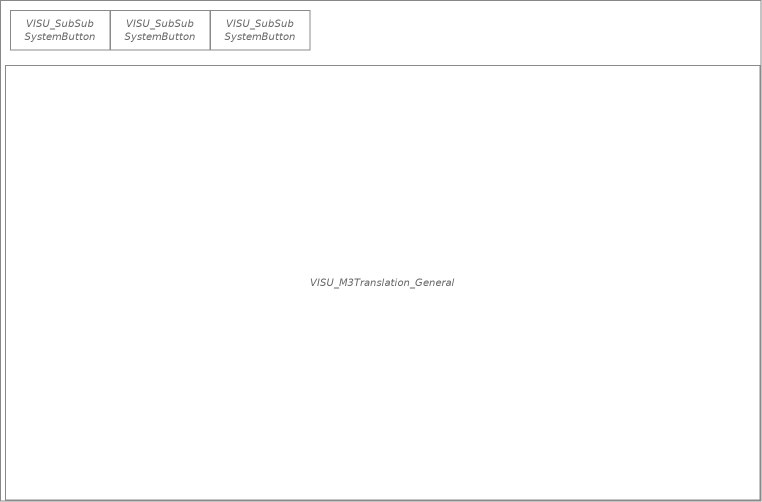
VISUALIZATION VISU_M3Translation  // 762x502
VAR_IN_OUT	
    ref : M3Translation;
    widget : M3TranslationWidget;
END_VAR
    Frame (5,65 755x435), frame switch variable: widget.activeTab
        shows VISU_M3Translation_General(ref := ref, widget := widget)
        shows VISU_LinearAxis(axis := ref.parts.motorAxis, widget := widget.motorAxis)
        shows VISU_FaulhaberDrive(drive := ref.parts.motorDrive, widget := widget.motorDrive)
        p3374720746: ref.parts.motorDrive
    Frame (10,10 100x40)
        shows VISU_SubSubSystemButton(widget := widget.button_general)
        OnMouseClick: FrameSelectionChange Selection=SelectedFrame=c1a27479-cf51-4fe2-b6d5-639dc505c4c1, GlobSel=AssignType=Directly, SelType=Locally
        OnMouseClick: execute { widget.activeTab := M3TranslationTabs.GENERAL; }
    Frame (110,10 100x40)
        shows VISU_SubSubSystemButton(widget := widget.button_axis)
        OnMouseClick: FrameSelectionChange Selection=SelectedFrame=c1a27479-cf51-4fe2-b6d5-639dc505c4c1, Selection=1, GlobSel=AssignType=Directly, SelType=Locally
        OnMouseClick: execute { widget.activeTab := M3TranslationTabs.AXIS; }
    Frame (210,10 100x40)
        shows VISU_SubSubSystemButton(widget := widget.button_drive)
        OnMouseClick: FrameSelectionChange Selection=SelectedFrame=c1a27479-cf51-4fe2-b6d5-639dc505c4c1, Selection=2, GlobSel=AssignType=Directly, SelType=Locally
        OnMouseClick: execute { widget.activeTab := M3TranslationTabs.DRIVE; }
END_VISUALIZATION

(* stored: Version 1.1.0.1, ProductVersion 3.1.4019.2
   Visu VISU_M3Translation: Id {ce46f2f0-5645-4c48-bfcc-35afac27e142} *)
